(* PLC project drive, Dassault Systèmes ControlBuild 2024x *)
(* stored: creationDateTime 2023-10-03T11:13:42-01:00 *)

PROGRAM bottling_line.drive
  VAR_INPUT
    autoMode : BOOL := false;
    manualMode : BOOL := false;
  END_VAR
  VAR_INPUT
    acknowledgePB : BOOL := false;
  END_VAR
  VAR_INPUT
    load : BOOL := false;
    evacuate : BOOL := false;
    convoy : BOOL := false;
  END_VAR
  VAR_INPUT
    inputFlow : REAL := 0.0;
  END_VAR
  VAR_OUTPUT
    bottlePresent : BOOL := false;
    bottleFilled : BOOL := false;
    pulse : BOOL := false;
  END_VAR

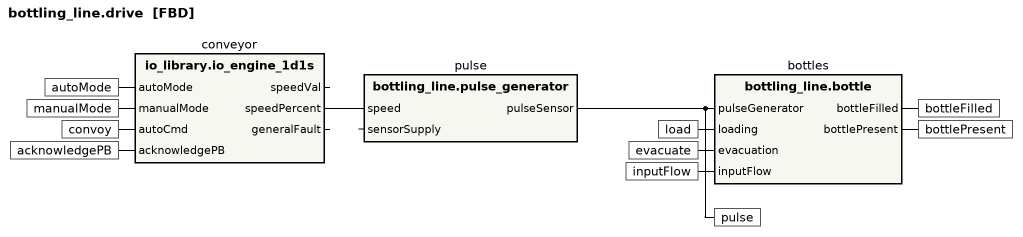
(* FBD diagram, written out as Structured Text *)
conveyor(autoMode := autoMode, manualMode := manualMode, autoCmd := convoy, acknowledgePB := acknowledgePB);
pulse(speed := conveyor.speedPercent);
pulse := pulse.pulseSensor;
bottles(pulseGenerator := pulse.pulseSensor, loading := load, evacuation := evacuate, inputFlow := inputFlow);
bottleFilled := bottles.bottleFilled;
bottlePresent := bottles.bottlePresent;
END_PROGRAM
